// Mitsubishi GX Works2 project: start_protect_stop   PLC: FX1S

PROGRAM MAIN
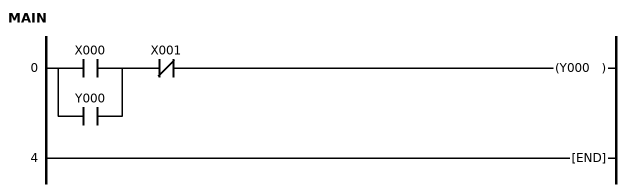
0     LD      X000
      OR      Y000
      ANI     X001
      OUT     Y000
4     END
END_PROGRAM
